FUNCTION_BLOCK TelemetryIO EXTENDS SM_TelemetryIO
VAR_INPUT
END_VAR
VAR_OUTPUT
END_VAR
VAR
    _testVar_TelemetryIO : BOOL;
END_VAR

SUPER^();

// do stuff

//SUPER^();

END_FUNCTION_BLOCK

(* stored: Version 1.1.0.1, ProductVersion 3.1.0.36
   POU TelemetryIO: Id {1137fc99-4890-47ef-9990-00b465da8fba}, SpecialFunc None *)
